FUNCTION_BLOCK FB_LED
VAR
	bInit : BOOL;
	Location : ARRAY[1..2] OF INT := [-1,-1];
	iNextUnit : I_NextUnit;
	iCurrentUnit : I_Unit;
	ForwardMoving : BOOL;
	fbTon : TON := (PT := T#1S);
	refCommand : REFERENCE TO E_Command;
END_VAR

IF NOT bInit OR Location[1] = -1 OR Location[2] = -1 THEN
	RETURN;
END_IF
ForwardMoving S= refCommand = E_Command.Forward;
ForwardMoving R= refCommand = E_Command.Backward;
IF iCurrentUnit.isStopped THEN
	fbTON(IN := FALSE);
	RETURN;
END_IF

IF NOT iCurrentUnit.LastLED OR ((iCurrentUnit <> 0 AND_THEN iCurrentUnit.isSendStart) AND (iNextUnit <> 0 AND_THEN iNextUnit.isReceiveStart))  THEN
	IF ForwardMoving THEN
		fbTon(IN := TRUE);
		IF fbTon.Q THEN
			fbTon(IN := FALSE);
			Location[1] := Location[1] + 1;
			Location[2] := Location[2] + 1;
		END_IF
	ELSE
		fbTon(IN := TRUE);
		IF fbTon.Q THEN
			fbTon(IN := FALSE);
			Location[1] := Location[1] - 1;
			Location[2] := Location[2] - 1;
		END_IF
	END_IF
ELSIF iNextUnit = 0 THEN
	fbTOn(IN := FALSE);
END_IF
Location[1] := LIMIT(0,Location[1],MAX_UNIT_NUMBER * 5 - 2);
Location[2] := LIMIT(0,Location[2],MAX_UNIT_NUMBER * 5 - 1);

METHOD GetFB_Unit
VAR_INPUT
	iCurrentUnit : I_Unit;
	iNextUnit : I_NextUnit;
END_VAR
THIS^.iCurrentUnit := iCurrentUnit;
THIS^.iNextUnit := iNextUnit;
END_METHOD

METHOD Initalize
VAR_IN_OUT
	refCommand : E_Command;
END_VAR
THIS^.refCommand REF= refCommand;
Location[1] := 0;
Location[2] := 1;
bInit := TRUE;
END_METHOD

PROPERTY Location1 : INT
GET
Location1 := Location[1];
END_GET
END_PROPERTY

PROPERTY Location2 : INT
GET
Location2 := Location[2];
END_GET
END_PROPERTY

METHOD Reset
VAR_INPUT
END_VAR
Location[1] := -1;
Location[2] := -1;
fbTON(IN := FALSE);
END_METHOD

END_FUNCTION_BLOCK

(* stored: Version 1.1.0.1, ProductVersion 3.1.4024.12
   POU FB_LED: Id {8405c9e3-492f-4f2f-8362-d43d0cf6a99c}, SpecialFunc None
   Method GetFB_Unit: Id {21a82efb-2475-42d2-bcc0-6fab990e2327}
   Method Initalize: Id {630be468-ab82-4cd5-a30a-e942c8713b61}
   Property Location1: Id {f6f2bd8f-c5e3-4198-8e48-4da8e6fbfa7d}
   Get Get: Id {454e022a-e897-4984-b25e-dce837b2a5b7}
   Property Location2: Id {b8fbf839-be0d-4d97-a449-515e51ef437a}
   Get Get: Id {2fd9b8e7-73f2-491b-95ca-451cd1c8f1f1}
   Method Reset: Id {5615a009-8261-4178-8dac-2720df089808} *)
